FUNCTION_BLOCK PID_Regler
VAR_INPUT
	R :			REAL;
	Y :			REAL;
	Modus :		System_Modus_Enum;
	Param :		PID_Parameter_Strukt;
	T :			REAL;
END_VAR
VAR_OUTPUT
END_VAR
VAR
END_VAR

CASE Modus OF
	System_Modus_Enum.System_Init:
	;
	System_Modus_Enum.System_Run:
	;
END_CASE

END_FUNCTION_BLOCK

(* stored: Version 1.1.0.1, ProductVersion 3.1.4024.13
   POU PID_Regler: Id {5a73cf8e-f42a-473f-9077-c1d965924ba7}, SpecialFunc None *)
